// TIA Portal project "Trabajo_68_Mejoras" (V15)

(* hardware
DEVICE "S7-1200 station_1"  S7-1200 Station
   slot 0: "Rack_0"  S7-1200 Rack  Rack  V1.0
   slot 1: "PLC_1"  CPU 1214C AC/DC/Rly  6ES7 214-1BG40-0XB0  V4.2
*)

// ===== PLC "PLC_1"  CPU 1214C AC/DC/Rly =====

VAR_GLOBAL   // PLC tag table "Tabla de variables estándar"
   "MI" AT %Q0.0 : Bool;
   "MD" AT %Q0.1 : Bool;
   "BI" AT %I0.0 : Bool;
   "BD" AT %I0.1 : Bool;
   "PI" AT %I0.2 : Bool;
   "PD" AT %I0.3 : Bool;
   "SI" AT %I0.4 : Bool;
   "SD" AT %I0.5 : Bool;
   "A" AT %Q0.2 : Bool;
   "C" AT %Q0.3 : Bool;
   "F" AT %I0.6 : Bool;
   "D" AT %I0.7 : Bool;
   "P" AT %I1.0 : Bool;
   "AB" AT %I1.1 : Bool;
   "PE" AT %I1.2 : Bool;
   "Mover derecha" AT %M0.0 : Bool;
   "Mover izquierda" AT %M0.1 : Bool;
   "Apertura puertas" AT %M0.2 : Bool;
   "Cierre puertas" AT %M0.3 : Bool;
   "Emergencia" AT %M0.4 : Bool;
   "CE" AT %I1.3 : Bool;
END_VAR

// folder: System blocks/Program resources

DATA_BLOCK "Temporizador 5s"   // DB1
{ S7_Optimized_Access := 'TRUE' }
AUTHOR : Simatic
FAMILY : IEC
NAME : IEC_TMR
VERSION : 1.0
// stored: InstanceOfName IEC_TIMER
"IEC_TIMER"
BEGIN
END_DATA_BLOCK

// folder: (top level)

ORGANIZATION_BLOCK "Main"   // OB1, LAD, ProgramCycle
TITLE = "Main Program Sweep (Cycle)"
{ S7_Optimized_Access := 'TRUE' }
VERSION : 0.1
   VAR_INPUT
      Initial_Call : Bool;   // Initial call of this OB
      Remanence : Bool;   // =True, if remanent data are available
   END_VAR
   VAR_TEMP   // added for the SCL form of the ladder/FBD networks
      _w1 : Bool;
      _w2 : Bool;
   END_VAR
BEGIN

REGION Network 1: Comprobaciones iniciales para Arranque normal
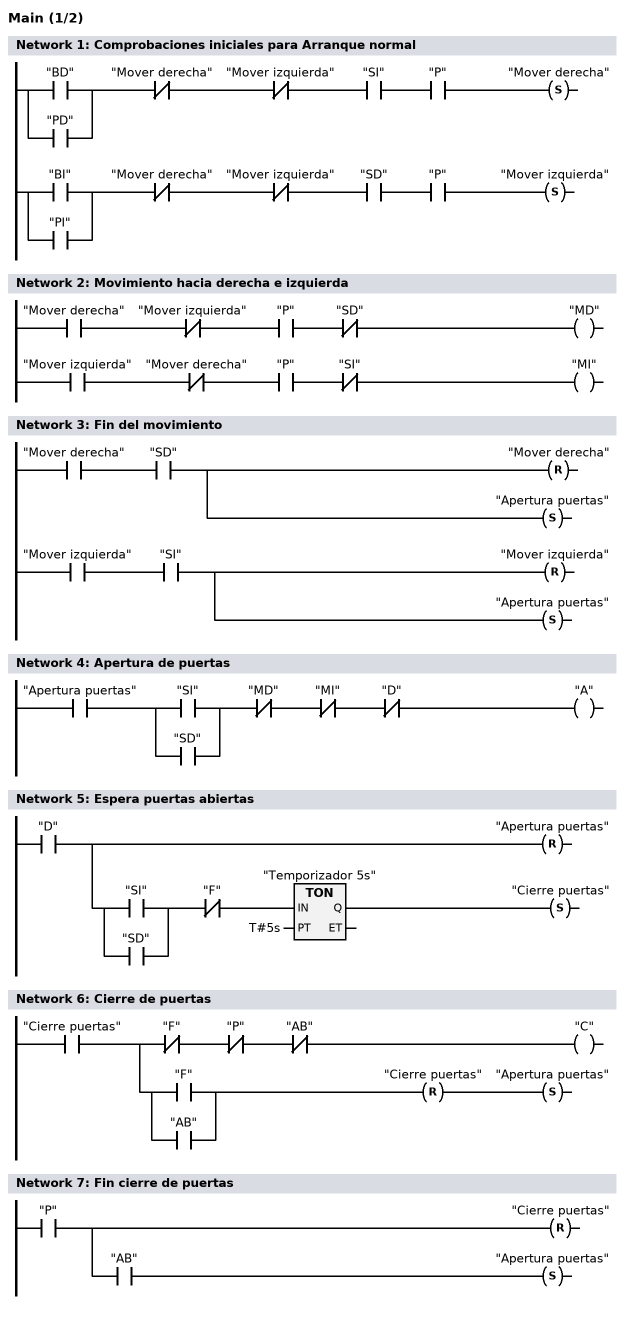
   RUNG wire#powerrail
      Contact( "BD" )
      wire#w1
      I_Contact( "Mover derecha" )
      I_Contact( "Mover izquierda" )
      Contact( "SI" )
      Contact( "P" )
      S_Coil( "Mover derecha" )
   END_RUNG
   RUNG wire#powerrail
      Contact( "PD" )
   END_RUNG wire#w1
   RUNG wire#powerrail
      Contact( "BI" )
      wire#w2
      I_Contact( "Mover derecha" )
      I_Contact( "Mover izquierda" )
      Contact( "SD" )
      Contact( "P" )
      S_Coil( "Mover izquierda" )
   END_RUNG
   RUNG wire#powerrail
      Contact( "PI" )
   END_RUNG wire#w2
   // the same network as SCL:
   IF ("BD" OR "PD") AND NOT "Mover derecha" AND NOT "Mover izquierda" AND "SI" AND "P" THEN
       "Mover derecha" := TRUE;
   END_IF;
   IF ("BI" OR "PI") AND NOT "Mover derecha" AND NOT "Mover izquierda" AND "SD" AND "P" THEN
       "Mover izquierda" := TRUE;
   END_IF;
END_REGION

REGION Network 2: Movimiento hacia derecha e izquierda
   RUNG wire#powerrail
      Contact( "Mover derecha" )
      I_Contact( "Mover izquierda" )
      Contact( "P" )
      I_Contact( "SD" )
      Coil( "MD" )
   END_RUNG
   RUNG wire#powerrail
      Contact( "Mover izquierda" )
      I_Contact( "Mover derecha" )
      Contact( "P" )
      I_Contact( "SI" )
      Coil( "MI" )
   END_RUNG
   // the same network as SCL:
   "MD" := "Mover derecha" AND NOT "Mover izquierda" AND "P" AND NOT "SD";
   "MI" := "Mover izquierda" AND NOT "Mover derecha" AND "P" AND NOT "SI";
END_REGION

REGION Network 3: Fin del movimiento
   RUNG wire#powerrail
      Contact( "Mover derecha" )
      Contact( "SD" )
      wire#w1
      R_Coil( "Mover derecha" )
   END_RUNG
   RUNG wire#w1
      S_Coil( "Apertura puertas" )
   END_RUNG
   RUNG wire#powerrail
      Contact( "Mover izquierda" )
      Contact( "SI" )
      wire#w2
      R_Coil( "Mover izquierda" )
   END_RUNG
   RUNG wire#w2
      S_Coil( "Apertura puertas" )
   END_RUNG
   // the same network as SCL:
   #_w1 := "Mover derecha" AND "SD";
   IF #_w1 THEN
       "Mover derecha" := FALSE;
       "Apertura puertas" := TRUE;
   END_IF;
   #_w2 := "Mover izquierda" AND "SI";
   IF #_w2 THEN
       "Mover izquierda" := FALSE;
       "Apertura puertas" := TRUE;
   END_IF;
END_REGION

REGION Network 4: Apertura de puertas
   RUNG wire#powerrail
      Contact( "Apertura puertas" )
      wire#w1
      Contact( "SI" )
      wire#w2
      I_Contact( "MD" )
      I_Contact( "MI" )
      I_Contact( "D" )
      Coil( "A" )
   END_RUNG
   RUNG wire#w1
      Contact( "SD" )
   END_RUNG wire#w2
   // the same network as SCL:
   "A" := "Apertura puertas" AND ("SI" OR "SD") AND NOT "MD" AND NOT "MI" AND NOT "D";
END_REGION

REGION Network 5: Espera puertas abiertas
   IF "D" THEN "Apertura puertas" := FALSE; END_IF;
   "Temporizador 5s".TON(IN := "D" AND ("SI" OR "SD") AND NOT "F", PT := T#5s);
   IF "Temporizador 5s".Q THEN "Cierre puertas" := TRUE; END_IF;
END_REGION

REGION Network 6: Cierre de puertas
   RUNG wire#powerrail
      Contact( "Cierre puertas" )
      wire#w1
      I_Contact( "F" )
      I_Contact( "P" )
      I_Contact( "AB" )
      Coil( "C" )
   END_RUNG
   RUNG wire#w1
      Contact( "F" )
      wire#w2
      R_Coil( "Cierre puertas" )
      S_Coil( "Apertura puertas" )
   END_RUNG
   RUNG wire#w1
      Contact( "AB" )
   END_RUNG wire#w2
   // the same network as SCL:
   "C" := "Cierre puertas" AND NOT "F" AND NOT "P" AND NOT "AB";
   #_w1 := "Cierre puertas" AND ("F" OR "AB");
   IF #_w1 THEN
       "Cierre puertas" := FALSE;
       "Apertura puertas" := TRUE;
   END_IF;
END_REGION

REGION Network 7: Fin cierre de puertas
   RUNG wire#powerrail
      Contact( "P" )
      wire#w1
      R_Coil( "Cierre puertas" )
   END_RUNG
   RUNG wire#w1
      Contact( "AB" )
      S_Coil( "Apertura puertas" )
   END_RUNG
   // the same network as SCL:
   IF "P" THEN "Cierre puertas" := FALSE; END_IF;
   IF "P" AND "AB" THEN "Apertura puertas" := TRUE; END_IF;
END_REGION

REGION Network 8: Parada de Emergencia
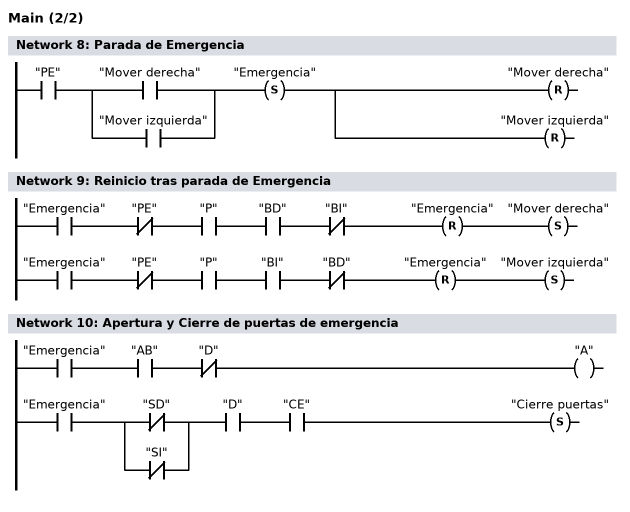
   RUNG wire#powerrail
      Contact( "PE" )
      wire#w1
      Contact( "Mover derecha" )
      wire#w2
      S_Coil( "Emergencia" )
      wire#w3
      R_Coil( "Mover derecha" )
   END_RUNG
   RUNG wire#w1
      Contact( "Mover izquierda" )
   END_RUNG wire#w2
   RUNG wire#w3
      R_Coil( "Mover izquierda" )
   END_RUNG
   // the same network as SCL:
   IF "PE" AND ("Mover derecha" OR "Mover izquierda") THEN "Emergencia" := TRUE; END_IF;
   #_w1 := "PE" AND ("Mover derecha" OR "Mover izquierda");
   IF #_w1 THEN
       "Mover derecha" := FALSE;
       "Mover izquierda" := FALSE;
   END_IF;
END_REGION

REGION Network 9: Reinicio tras parada de Emergencia
   RUNG wire#powerrail
      Contact( "Emergencia" )
      I_Contact( "PE" )
      Contact( "P" )
      Contact( "BD" )
      I_Contact( "BI" )
      R_Coil( "Emergencia" )
      S_Coil( "Mover derecha" )
   END_RUNG
   RUNG wire#powerrail
      Contact( "Emergencia" )
      I_Contact( "PE" )
      Contact( "P" )
      Contact( "BI" )
      I_Contact( "BD" )
      R_Coil( "Emergencia" )
      S_Coil( "Mover izquierda" )
   END_RUNG
   // the same network as SCL:
   #_w1 := "Emergencia" AND NOT "PE" AND "P" AND "BD" AND NOT "BI";
   IF #_w1 THEN
       "Emergencia" := FALSE;
       "Mover derecha" := TRUE;
   END_IF;
   #_w2 := "Emergencia" AND NOT "PE" AND "P" AND "BI" AND NOT "BD";
   IF #_w2 THEN
       "Emergencia" := FALSE;
       "Mover izquierda" := TRUE;
   END_IF;
END_REGION

REGION Network 10: Apertura y Cierre de puertas de emergencia
   RUNG wire#powerrail
      Contact( "Emergencia" )
      Contact( "AB" )
      I_Contact( "D" )
      Coil( "A" )
   END_RUNG
   RUNG wire#powerrail
      Contact( "Emergencia" )
      wire#w1
      I_Contact( "SD" )
      wire#w2
      Contact( "D" )
      Contact( "CE" )
      S_Coil( "Cierre puertas" )
   END_RUNG
   RUNG wire#w1
      I_Contact( "SI" )
   END_RUNG wire#w2
   // the same network as SCL:
   "A" := "Emergencia" AND "AB" AND NOT "D";
   IF "Emergencia" AND (NOT "SD" OR NOT "SI") AND "D" AND "CE" THEN "Cierre puertas" := TRUE; END_IF;
END_REGION
END_ORGANIZATION_BLOCK